FUNCTION_BLOCK TransLeftCheck (* Template for a Basic Function Block Type *)
  (* Standard: 61499-2 *)
  (* Version 1.0, 2021-07-28, Tuojian Lyu *)
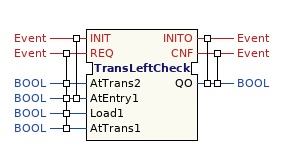
  EVENT_INPUT
    INIT WITH AtEntry1; (* Initialization Request *)
    REQ WITH AtEntry1, Load1, AtTrans2, AtTrans1; (* Normal Execution Request *)
  END_EVENT
  EVENT_OUTPUT
    INITO WITH QO; (* Initialization Confirm *)
    CNF WITH QO; (* Execution Confirmation *)
  END_EVENT
  VAR_INPUT
    AtTrans2 : BOOL;
    AtEntry1 : BOOL; (* Input event qualifier *)
    Load1 : BOOL;
    AtTrans1 : BOOL;
  END_VAR
  VAR_OUTPUT
    QO : BOOL; (* Output event qualifier *)
  END_VAR
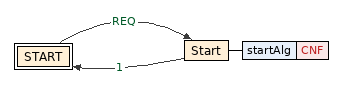
  EC_STATES
    START; (* Initial State *)
    Start : startAlg -> CNF;
  END_STATES
  EC_TRANSITIONS
    START TO Start := REQ;
    Start TO START := 1;
  END_TRANSITIONS
  ALGORITHM startAlg IN ST:
IF (FALSE = QO) AND (TRUE = AtTrans2) THEN
QO := TRUE;
END_IF;

IF (TRUE = QO) AND (TRUE = AtTrans1) THEN
QO := FALSE;
END_IF;

IF (TRUE = AtEntry1) THEN
QO := FALSE;
END_IF;
  END_ALGORITHM
END_FUNCTION_BLOCK
